KUKA KRL program: AirSensorSps.src, AirSensorSps.dat

--- AirSensorSps.src ---
&ACCESS RV
&REL 154
&COMMENT Ansteuerung Micromaster Frequenzumrichter
&PARAM EDITMASK = *
&PARAM TEMPLATE = C:\KRC\Roboter\Template\ExpertSubmit
DEF AirSensorSps( _bFault:OUT  )

;************************************************
;              CNC Robotics Ltd
;              Unit 3
;              www.cncrobotics.co.uk
;************************************************
;     Contact: helpdesk@cncrobotics.co.uk
;     Date: 05/04/24
;     Version: 1.17.54
;************************************************
; Description: sps control specific for the spindle.
;************************************************

ENUM SYSYEM_STATE _systemState
BOOL _bFault

IF (NOT iAirOK) THEN
    _bFault = TRUE
ELSE
    _bFault=FALSE
ENDIF


END

--- AirSensorSps.dat ---
&ACCESS  RV
&COMMENT Ansteuerung Micromaster Frequenzumrichter
&PARAM EDITMASK = *
&PARAM TEMPLATE = C:\KRC\Roboter\Template\ExpertSubmit
&PARAM TEMPLATE = C:\KRC\Roboter\Template\ExpertSubmit
&REL 154
DEFDAT  AIRSENSORSPS PUBLIC

;To Be included in the CNCRSignals Folder
;digital inputs
;GLOBAL SIGNAL iAirOK $IN[1] ;Air ok pressure switch


GLOBAL BOOL bAirMessage=TRUE ;for triggering air message
GLOBAL BOOL bAirInterrupt=FALSE ; Interrupt Flag when a problem with air messages
GLOBAL BOOL bAirConfirmed=FALSE
ENDDAT
